// TwinCAT 3 PLC project Untitled1
// ProgramVersion: 3.1.4024.0
// libraries:
//   Tc2_Standard, * (Beckhoff Automation GmbH)
//   Tc2_System, * (Beckhoff Automation GmbH)
//   Tc2_Utilities, * (Beckhoff Automation GmbH)
//   Tc3_Module, * (Beckhoff Automation GmbH)
// project tree:
//   / PlcTask.TcTTO
//   POUs/ MAIN.TcPOU
// real-time tasks:
//   TASK Task 1: cycle T#10ms, priority 1, ADS port 350
//   TASK PlcTask: cycle T#10ms, priority 20, ADS port 351
// variable links:
//   Untitled1/Untitled1 Instance <-> TrackRtStartTime/TrackRtStartTime_Obj1 (RtStartTimeModule)
//     PlcTask Inputs/MAIN.t_startTimeRt <-> Outputs/RtStartTime

CONFIGURATION Untitled1
    RESOURCE PLC ON TwinCAT3
        TASK PlcTask(INTERVAL := T#10ms, PRIORITY := 20);
        PROGRAM MAIN WITH PlcTask : MAIN;
    END_RESOURCE
END_CONFIGURATION

// ---- POUs/MAIN.TcPOU
PROGRAM MAIN
VAR
	t_startTimeRt AT %I* :ULINT; 
	rtStartTime : TIMESTRUCT;
	b_convert : BOOL;
END_VAR

IF b_convert THEN
	rtStartTime := DT_TO_SYSTEMTIME(FILETIME64_TO_DT(t_startTimeRt));
END_IF

END_PROGRAM
